FUNCTION_BLOCK F_ADD (* Adding two values *)
  (* Standard: 61499-1; Description: Copyright (c) 2023 Johannes Kepler University Linz This program and the accompanying materials are made available under the terms of the Eclipse Public License 2.0 which is available at https://www.eclipse.org/legal/epl-2.0/ SPDX-License-Identifier: EPL-2.0 *)
  (* Version 1.0, 2023-03-07, Bianca Wiesmayr, Johannes Kepler University Linz, initial API and implementation and/or initial documentation *)
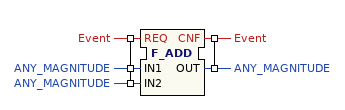
  EVENT_INPUT
    REQ WITH IN1, IN2; (* Normal Execution Request *)
  END_EVENT
  EVENT_OUTPUT
    CNF WITH OUT; (* Execution Confirmation *)
  END_EVENT
  VAR_INPUT
    IN1 : ANY_MAGNITUDE;
    IN2 : ANY_MAGNITUDE;
  END_VAR
  VAR_OUTPUT
    OUT : ANY_MAGNITUDE;
  END_VAR
  ALGORITHM REQ IN ST:
VAR_TEMP
	X : LREAL;
	Y : LREAL;
END_VAR
	X := IN1;
	Y := IN2;
	OUT := X + Y;
  END_ALGORITHM
END_FUNCTION_BLOCK
